// TIA Portal V19 export
TYPE "LEXCHANGETRAY_typeNgConveyorEm_interface"
// stored: Access Published
   STRUCT
      deliver : "LEXCHANGETRAY_typeNgConveyor_deliver_interface";
      recieve : "LEXCHANGETRAY_typeNgConveyorEm_recieve_interface";
   END_STRUCT;
END_TYPE
